FUNCTION Convert_DATE_TO_BYTE : Hresult
VAR_INPUT
	in : DATE;
	out : REFERENCE TO BYTE;
END_VAR
VAR
	converted : BYTE;
END_VAR

converted := DATE_TO_BYTE(in);

IF (BYTE_TO_DATE(converted) <> in) THEN
	Convert_DATE_TO_BYTE := INCOMPATIBLE;
	RETURN;
END_IF

out := converted;

END_FUNCTION

(* stored: Version 1.1.0.1, ProductVersion 3.1.4024.12
   POU Convert_DATE_TO_BYTE: Id {2baf8031-724a-4999-ad16-17a33081a2e9}, SpecialFunc None *)
